INTERFACE IStirBlock

PROPERTY pEndFeedback : BOOL
GET
END_GET
END_PROPERTY

PROPERTY pStartFeedback : BOOL
GET
END_GET
END_PROPERTY

METHOD Stir : BOOL
VAR_INPUT
	sTargetName : STRING;
	bStirStartCommand : BOOL;
	bStirEndCommand : BOOL;
	nStirSetPoint : INT;
END_VAR
END_METHOD

END_INTERFACE

(* stored: Version 1.1.0.1, ProductVersion 3.1.4024.6
   Itf IStirBlock: Id {c17dbb49-032c-44b2-90e7-d518fc69893c}
   Property pEndFeedback: Id {744fb7d2-aa5b-4cc0-9c56-55c9b30d5a7b}
   Get Get: Id {3256aeb7-a26a-47a2-9f6c-7a650b828995}
   Property pStartFeedback: Id {a894cdd6-2f2d-4054-a465-b216ed6054ef}
   Get Get: Id {cffad5f0-460e-4e8e-b8e1-5267934251e9}
   Method Stir: Id {708211cb-132d-4d88-ad06-c7e31eb209be} *)
